(* PLC project Unnamed, Unknown Unnamed 1 *)
(* stored: creationDateTime 2022-06-03T13:37:24, modificationDateTime 2023-02-19T01:36:55 *)

PROGRAM ConveyorV1
  VAR
    StartButton AT %IX100.0 : BOOL;
    SafeDoor AT %IX100.1 : BOOL;
    Box_Not_Waiting AT %IX100.2 : BOOL;
    Picker_Holding AT %IX100.3 : BOOL;
    Picker_Rotating AT %IX100.4 : BOOL;
    Picker_Moving_Z AT %IX100.5 : BOOL;
    Conveyor_Move AT %QX100.0 : BOOL;
    Picker_Move_Down AT %QX100.1 : BOOL;
    Picker_Grab AT %QX100.2 : BOOL;
    Picker_Rotate_CCW AT %QX100.3 : BOOL;
    Picker_Rotate_CW AT %QX100.4 : BOOL;
  END_VAR
  VAR
    RUN : BOOL;
  END_VAR
  VAR  (* added by the conversion: wires and edge detectors of the diagram *)
    F_TRIG1 : F_TRIG;
    R_TRIG2 : R_TRIG;
    F_TRIG3 : F_TRIG;
    F_TRIG4 : F_TRIG;
  END_VAR

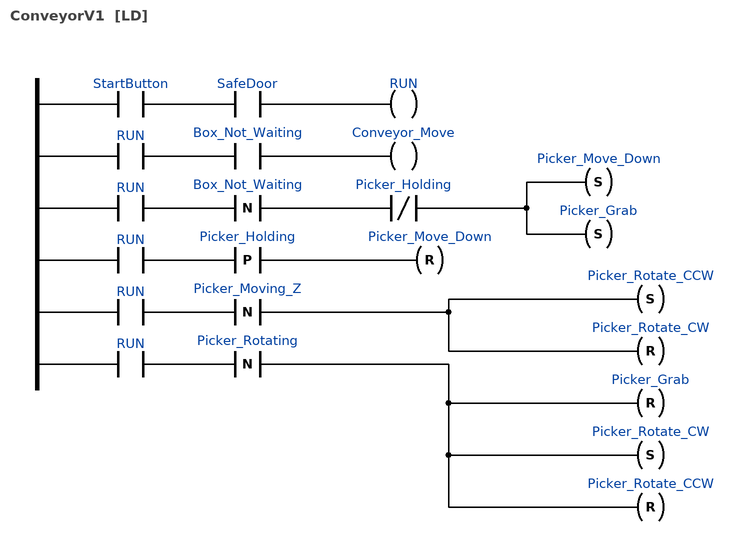
(* LD diagram, written out as Structured Text *)
RUN := StartButton AND SafeDoor;
Conveyor_Move := RUN AND Box_Not_Waiting;
F_TRIG1(CLK := Box_Not_Waiting);
IF RUN AND F_TRIG1.Q AND NOT Picker_Holding THEN Picker_Move_Down := TRUE; END_IF;
IF RUN AND F_TRIG1.Q AND NOT Picker_Holding THEN Picker_Grab := TRUE; END_IF;
R_TRIG2(CLK := Picker_Holding);
IF RUN AND R_TRIG2.Q THEN Picker_Move_Down := FALSE; END_IF;
F_TRIG3(CLK := Picker_Moving_Z);
IF RUN AND F_TRIG3.Q THEN Picker_Rotate_CCW := TRUE; END_IF;
IF RUN AND F_TRIG3.Q THEN Picker_Rotate_CW := FALSE; END_IF;
F_TRIG4(CLK := Picker_Rotating);
IF RUN AND F_TRIG4.Q THEN Picker_Grab := FALSE; END_IF;
IF RUN AND F_TRIG4.Q THEN Picker_Rotate_CW := TRUE; END_IF;
IF RUN AND F_TRIG4.Q THEN Picker_Rotate_CCW := FALSE; END_IF;
END_PROGRAM

CONFIGURATION Config0
  RESOURCE Res0 ON PLC
    TASK task0(INTERVAL := T#20ms, PRIORITY := 0);
    PROGRAM instance0 WITH task0 : ConveyorV1;
  END_RESOURCE
END_CONFIGURATION
